// TwinCAT 3 PLC project PLCStudent
// ProgramVersion: 3.1.4022.3
// libraries:
//   Tc2_Standard, * (Beckhoff Automation GmbH)
//   Tc2_System, * (Beckhoff Automation GmbH)
//   Tc3_Module, * (Beckhoff Automation GmbH)
// project tree:
//   GVLs/ GVL.TcGVL
//   / PlcTask.TcTTO
//   POUs/ Auto_Manual.TcPOU, Emergency_Stop.TcPOU, Auto_Mode.TcPOU, MAIN.TcPOU
// (motion and I/O tree: see PLC project plcsim)
// real-time tasks:
//   TASK PlcTask: cycle T#30ms, priority 20, ADS port 350
// variable links:
//   PLCSim/PLCSim Instance <-> PLCStudent/PLCStudent Instance
//     PlcTask Inputs/MAIN.ixDrillDown <-> PlcTask Outputs/GVL.qxDrillDown
//     PlcTask Inputs/MAIN.ixDrillUp <-> PlcTask Outputs/GVL.qxDrillUp
//     PlcTask Inputs/MAIN.ixLampEmStopOk <-> PlcTask Outputs/GVL.qxLampEmStopOk
//     PlcTask Inputs/MAIN.ixLampHomePos <-> PlcTask Outputs/GVL.qxLampHomePos
//     PlcTask Inputs/MAIN.ixLampSafetyOk <-> PlcTask Outputs/GVL.qxLampSafetyOk
//     PlcTask Inputs/MAIN.ixLampStarted <-> PlcTask Outputs/GVL.qxGreenLamp
//     PlcTask Inputs/MAIN.ixSliderAin <-> PlcTask Outputs/GVL.qxAin
//     PlcTask Inputs/MAIN.ixSliderAout <-> PlcTask Outputs/GVL.qxAout
//     PlcTask Inputs/MAIN.ixSliderBin <-> PlcTask Outputs/GVL.qxBin
//     PlcTask Inputs/MAIN.ixSliderBout <-> PlcTask Outputs/GVL.qxBout
//     PlcTask Outputs/MAIN.nCnt <-> PlcTask Inputs/GVL.iwCounter
//     PlcTask Outputs/MAIN.qsOrderNum <-> PlcTask Inputs/GVL.iwOrderNum
//     PlcTask Outputs/MAIN.qxAuto <-> PlcTask Inputs/GVL.ixAuto
//     PlcTask Outputs/MAIN.qxBtn1EmStopOk <-> PlcTask Inputs/GVL.ixBtn1EmStopOk
//     PlcTask Outputs/MAIN.qxBtn2EmStopOk <-> PlcTask Inputs/GVL.ixBtn2EmStopOk
//     PlcTask Outputs/MAIN.qxBtnAin <-> PlcTask Inputs/GVL.ixBtnAin
//     PlcTask Outputs/MAIN.qxBtnAout <-> PlcTask Inputs/GVL.ixBtnAout
//     PlcTask Outputs/MAIN.qxBtnBin <-> PlcTask Inputs/GVL.ixBtnBin
//     PlcTask Outputs/MAIN.qxBtnBout <-> PlcTask Inputs/GVL.ixBtnBout
//     PlcTask Outputs/MAIN.qxBtnDrillIn <-> PlcTask Inputs/GVL.ixBtnDrillIn
//     PlcTask Outputs/MAIN.qxBtnDrillOut <-> PlcTask Inputs/GVL.ixBtnDrillOut
//     PlcTask Outputs/MAIN.qxBtnReset <-> PlcTask Inputs/GVL.ixBtnReset
//     PlcTask Outputs/MAIN.qxButtonStart <-> PlcTask Inputs/GVL.ixStart
//     PlcTask Outputs/MAIN.qxButtonStop <-> PlcTask Inputs/GVL.ixStop
//     PlcTask Outputs/MAIN.qxDrillDown <-> PlcTask Inputs/GVL.ixDrillDown
//     PlcTask Outputs/MAIN.qxDrillUp <-> PlcTask Inputs/GVL.ixDrillUp
//     PlcTask Outputs/MAIN.qxSafety1StopOk <-> PlcTask Inputs/GVL.ixSafety1StopOk
//     PlcTask Outputs/MAIN.qxSafety2StopOk <-> PlcTask Inputs/GVL.ixSafety2StopOk
//     PlcTask Outputs/MAIN.qxSliderAin <-> PlcTask Inputs/GVL.ixAin
//     PlcTask Outputs/MAIN.qxSliderAout <-> PlcTask Inputs/GVL.ixAout
//     PlcTask Outputs/MAIN.qxSliderBin <-> PlcTask Inputs/GVL.ixBin
//     PlcTask Outputs/MAIN.qxSliderBout <-> PlcTask Inputs/GVL.ixBout

CONFIGURATION PLCStudent
    RESOURCE PLC ON TwinCAT3
        TASK PlcTask(INTERVAL := T#30ms, PRIORITY := 20);
        PROGRAM MAIN WITH PlcTask : MAIN;
    END_RESOURCE
END_CONFIGURATION

// ---- GVLs/GVL.TcGVL
{attribute 'qualified_only'}
VAR_GLOBAL
	qxGreenLamp		AT %Q* : BOOL;
	qxAout		 	AT %Q* : BOOL; 
	qxAin 			AT %Q* : BOOL; 
	qxBout		 	AT %Q* : BOOL; 
	qxBin 			AT %Q* : BOOL; 
	qxDrillDown 	AT %Q* : BOOL;
	qxDrillUp		AT %Q* : BOOL;
	qxLampEmStopOk	AT %Q* : BOOL;
	qxLampSafetyOk  AT %Q* : BOOL;
	qxLampHomePos   AT %Q* : BOOL;
	
	
	ixStart			AT %I* : BOOL;
	ixStop			AT %I* : BOOL;
	ixAout			AT %I* : BOOL;
	ixAin			AT %I* : BOOL;
	ixBout			AT %I* : BOOL;
	ixBin			AT %I* : BOOL;
	ixDrillUp		AT %I* : BOOL;
	ixDrillDown		AT %I* : BOOL;

	ixAuto			AT %I* : BOOL;
	ixBtn1EmStopOk	AT %I* : BOOL;
	ixBtn2EmStopOk	AT %I* : BOOL;	
	ixSafety1StopOk	AT %I* : BOOL;
	ixSafety2StopOk	AT %I* : BOOL;	
	ixBtnReset		AT %I* : BOOL;
	ixBtnAout		AT %I* : BOOL;
	ixBtnAin		AT %I* : BOOL;
	ixBtnBout		AT %I* : BOOL;
	ixBtnBin		AT %I* : BOOL;
	ixBtnDrillOut	AT %I* : BOOL;
	ixBtnDrillIn	AT %I* : BOOL;
	iwCounter		AT %I*	:INT;
	iwOrderNum		AT %I*	:INT;
END_VAR

// ---- POUs/MAIN.TcPOU
PROGRAM MAIN
VAR
END_VAR

Auto_Manual();
Emergency_Stop();

END_PROGRAM

// ---- POUs/Auto_Manual.TcPOU
PROGRAM Auto_Manual
VAR
END_VAR

IF gvl.ixAuto THEN
	Auto_Mode();	
END_IF

END_PROGRAM

// ---- POUs/Auto_Mode.TcPOU
PROGRAM Auto_Mode
VAR_INPUT
	SFCPause:BOOL;
	SFCCurrentStep:STRING;
	SFCInit:BOOL;
END_VAR
VAR
	Activator: INT;
END_VAR

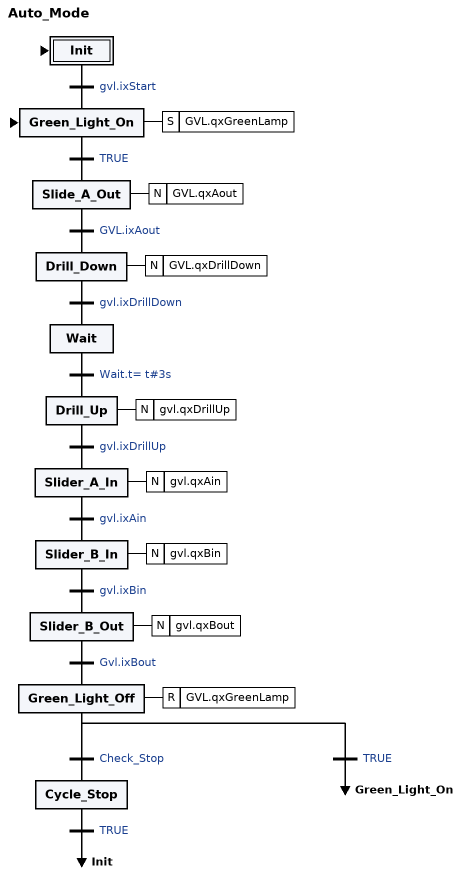
INITIAL_STEP Init:
END_STEP
TRANSITION FROM Init TO Green_Light_On
    := gvl.ixStart;
END_TRANSITION
STEP Green_Light_On:
    GVL.qxGreenLamp(S);
END_STEP
TRANSITION FROM Green_Light_On TO Slide_A_Out
    := TRUE;
END_TRANSITION
STEP Slide_A_Out:
    GVL.qxAout(N);
END_STEP
TRANSITION FROM Slide_A_Out TO Drill_Down
    := GVL.ixAout;
END_TRANSITION
STEP Drill_Down:
    GVL.qxDrillDown(N);
END_STEP
TRANSITION FROM Drill_Down TO Wait
    := gvl.ixDrillDown;
END_TRANSITION
STEP Wait:
END_STEP
TRANSITION FROM Wait TO Drill_Up
    := Wait.t= t#3s;
END_TRANSITION
STEP Drill_Up:
    gvl.qxDrillUp(N);
END_STEP
TRANSITION FROM Drill_Up TO Slider_A_In
    := gvl.ixDrillUp;
END_TRANSITION
STEP Slider_A_In:
    gvl.qxAin(N);
END_STEP
TRANSITION FROM Slider_A_In TO Slider_B_In
    := gvl.ixAin;
END_TRANSITION
STEP Slider_B_In:
    gvl.qxBin(N);
END_STEP
TRANSITION FROM Slider_B_In TO Slider_B_Out
    := gvl.ixBin;
END_TRANSITION
STEP Slider_B_Out:
    gvl.qxBout(N);
END_STEP
TRANSITION FROM Slider_B_Out TO Green_Light_Off
    := Gvl.ixBout;
END_TRANSITION
STEP Green_Light_Off:
    GVL.qxGreenLamp(R);
END_STEP
TRANSITION FROM Green_Light_Off TO Cycle_Stop
    := Check_Stop;
END_TRANSITION
STEP Cycle_Stop:
END_STEP
TRANSITION FROM Cycle_Stop TO Init
    := TRUE;
END_TRANSITION
TRANSITION FROM Green_Light_Off TO Green_Light_On
    := TRUE;
END_TRANSITION

TRANSITION Check_Stop:
IF gvl.ixStop THEN
	Activator:= 1;
END_IF
IF Activator=1 THEN
	Check_Stop:=TRUE;
END_IF
IF gvl.ixStart THEN
	Activator:= 0;
	Check_Stop:=FALSE;
END_IF
END_TRANSITION

END_PROGRAM

// ---- POUs/Emergency_Stop.TcPOU
PROGRAM Emergency_Stop
VAR
END_VAR

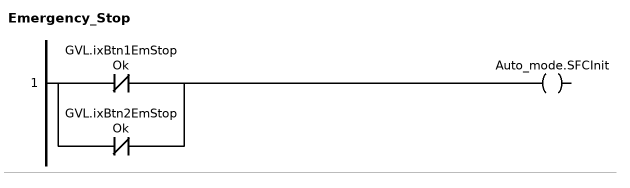
// NETWORK 1
Auto_mode.SFCInit := NOT GVL.ixBtn1EmStopOk OR NOT GVL.ixBtn2EmStopOk;

END_PROGRAM
